TYPE ST_Machine_Command :
	STRUCT
		StartHoming : BOOL;
	END_STRUCT
END_TYPE

(* stored: Version 1.1.0.1
   DUT ST_Machine_Command: Id {26415c7a-814b-4a50-8bac-47e7087a13e6} *)
